// TwinCAT 3 PLC project mini_powermeter_calib
// ProgramVersion: 3.1.4022.7
// libraries:
//   LCLS General, * (SLAC)
//   lcls-twincat-motion, * (SLAC)
//   lcls2-cc-lib, * (SLAC)
//   PMPS, * (SLAC - LCLS)
//   Tc2_Standard, * (Beckhoff Automation GmbH)
//   Tc2_System, * (Beckhoff Automation GmbH)
//   Tc3_Module, * (Beckhoff Automation GmbH)
// project tree:
//   / GlobalTextList.TcGTLO, PlcTask.TcTTO
//   GVLs/ GVL.TcGVL, Main.TcGVL
//   POUs/ FB_AnalogInput_DINT.TcPOU, FB_PPM_PowerMeter_DINT.TcPOU, PRG_MAIN.TcPOU, PRG_IM1_PPM.TcPOU, PRG_IM2_PPM.TcPOU
// real-time tasks:
//   TASK PlcTask: cycle T#10ms, priority 20, ADS port 350
//   TASK VISU_TASK: cycle T#200000us, priority 30, ADS port 351
// motion (NC):
//   TASK NC-Task 1 SAF: cycle T#2ms, priority 4, ADS port 501
//   TASK NC-Task 1 SVB: cycle T#10ms, priority 8, ADS port 511
//   AXIS Axis 1 IM1TST-PPM-MMS (id 1)
//     Dynamic: AccelerationMaximum=200, DecelerationMaximum=200, Acceleration=200, Deceleration=200, Jerk=1000, DelayTime=0.004
//     Velo: Maximum=65
//     MotionControl: Enable=true, Range=0.0005, Time=1
//     TargetPosControl: Range=0.01, Time=1
//     OtherSettings: AllowMotionCmdToSlave=true
//     encoder EncType=29
//       EncPara: ScaleFactorNumerator=5e-05, Offset=-214686.941, MaxCount=#xffffffff, MaxCountHighDWord=#x0000001f
//         SoftEndMinControl: Enable=true, Range=-101.12
//         SoftEndMaxControl: Enable=true, Range=-11
//         Inc: RefSoftSyncMask=#x0000ffff
//     drive DrvType=24
//       Analog: VeloReferenz=100, ScaleFactorActTorque=0.1
//       TimeComp: TaskDelayCycles=1
//     controller CtrType=2
//       CtrPara: PriorControlFactor=1
//         PosDiffControl: Range=10, Time=0.1
//         PID: PosKp=10, PosExtKp=0.01, PosExtVelo=0.0005, DeadBandPosition=0.0001
//         Observer: BandWidth=20
//   AXIS Axis 2 IM2TST-PPM-MMS (id 23)
//     Dynamic: AccelerationMaximum=200, DecelerationMaximum=200, Acceleration=200, Deceleration=200, Jerk=1000, DelayTime=0.004
//     Velo: Maximum=65
//     MotionControl: Enable=true, Range=0.0005, Time=1
//     TargetPosControl: Range=0.01, Time=1
//     OtherSettings: AllowMotionCmdToSlave=true
//     encoder EncType=29
//       EncPara: ScaleFactorNumerator=5e-05, Offset=-214686.941, MaxCount=#xffffffff, MaxCountHighDWord=#x0000001f
//         SoftEndMinControl: Enable=true, Range=-101.12
//         SoftEndMaxControl: Enable=true, Range=-11
//         Inc: RefSoftSyncMask=#x0000ffff
//     drive DrvType=24
//       Analog: VeloReferenz=100, ScaleFactorActTorque=0.1
//       TimeComp: TaskDelayCycles=1
//     controller CtrType=2
//       CtrPara: PriorControlFactor=1
//         PosDiffControl: Range=10, Time=0.1
//         PID: PosKp=10, PosExtKp=0.01, PosExtVelo=0.0005, DeadBandPosition=0.0001
//         Observer: BandWidth=20
// I/O:
//   DEVICE Device 1 (EtherCAT), AmsNetId 172.21.148.90.2.1
//     Term 1 (EK1200) [EK1200-5000 EtherCAT Power supply (2A E-Bus)]
//       Term 2 (EL3602) [EL3602 2Ch. Ana. Input +/-10Volt, Diff. 24bit]
//       Term 3 (EK1122) [EK1122 2 port EtherCAT junction]
//         X1 IM1-PPM (EK1100) [EK1100 EtherCAT Coupler (2A E-Bus)]
//           IM1-EL7041 [EL7041 1Ch. Stepper motor output stage (50V, 5A)]
//           IM1-EL5042 [EL5042 2Ch. BiSS-C Encoder]
//           IM1-EL2004 [EL2004 4Ch. Dig. Output 24V, 0.5A]
//           IM1-EL3314 [EL3314 4Ch. Ana. Input Thermocouple (TC)]
//           IM1-EL3052 [EL3052 2Ch. Ana. Input 4-20mA]
//           IM1-EL3062 [EL3062 2Ch. Ana. Input 0-10V]
//           IM1-EL4004 [EL4004 4Ch. Ana. Output 0-10V, 12bit]
//           IM1-EL9011
//         X2 IM2-PPM (EK1100) [EK1100 EtherCAT Coupler (2A E-Bus)]
//           IM2-EL7041 [EL7041 1Ch. Stepper motor output stage (50V, 5A)]
//           IM2-EL5042 [EL5042 2Ch. BiSS-C Encoder]
//           IM2-EL2004 [EL2004 4Ch. Dig. Output 24V, 0.5A]
//           IM2-EL3314 [EL3314 4Ch. Ana. Input Thermocouple (TC)]
//           IM2-EL3052 [EL3052 2Ch. Ana. Input 4-20mA]
//           IM2-EL3062 [EL3062 2Ch. Ana. Input 0-10V]
//           IM2-EL4004 [EL4004 4Ch. Ana. Output 0-10V, 12bit]
//           IM2-EL9011 [EL9011 End Terminal]
//       Term 4 (EL9011) [EL9011 End Terminal]
// variable links:
//   (this object) <-> Device 1 (EtherCAT)/Term 1 (EK1200)/Term 3 (EK1122)/X1 IM1-PPM (EK1100)/IM1-EL5042
//     Enc/Inputs/In/nComState @bit 1 <-> WcState/InputToggle
//     Enc/Inputs/In/nComState <-> WcState/WcState
//     Enc/Inputs/In/nDataIn1 <-> FB Inputs Channel 1/Position
//     Enc/Inputs/In/nState1 @bit 12 <-> FB Inputs Channel 1/Status/Diag
//     Enc/Inputs/In/nState1 @bit 1 <-> FB Inputs Channel 1/Status/Error
//     Enc/Inputs/In/nState1 @bit 14 <-> FB Inputs Channel 1/Status/Input cycle counter
//     Enc/Inputs/In/nState1 @bit 2 <-> FB Inputs Channel 1/Status/Ready
//     Enc/Inputs/In/nState1 @bit 13 <-> FB Inputs Channel 1/Status/TxPDO State
//     Enc/Inputs/In/nState1 <-> FB Inputs Channel 1/Status/Warning
//   (this object) <-> Device 1 (EtherCAT)/Term 1 (EK1200)/Term 3 (EK1122)/X1 IM1-PPM (EK1100)/IM1-EL7041
//     Drive/Inputs/In/nState1 @bit 3 <-> STM Status/Status/Error
//     Drive/Inputs/In/nState1 @bit 5 <-> STM Status/Status/Moving negative
//     Drive/Inputs/In/nState1 @bit 4 <-> STM Status/Status/Moving positive
//     Drive/Inputs/In/nState1 @bit 1 <-> STM Status/Status/Ready
//     Drive/Inputs/In/nState1 <-> STM Status/Status/Ready to enable
//     Drive/Inputs/In/nState1 @bit 6 <-> STM Status/Status/Torque reduced
//     Drive/Inputs/In/nState1 @bit 2 <-> STM Status/Status/Warning
//     Drive/Inputs/In/nState2 @bit 3 <-> STM Status/Status/Digital input 1
//     Drive/Inputs/In/nState2 @bit 4 <-> STM Status/Status/Digital input 2
//     Drive/Inputs/In/nState2 @bit 5 <-> STM Status/Status/Sync error
//     Drive/Inputs/In/nState2 @bit 7 <-> STM Status/Status/TxPDO Toggle
//     Drive/Inputs/In/nState4 @bit 1 <-> WcState/InputToggle
//     Drive/Inputs/In/nState4 <-> WcState/WcState
//     Drive/Outputs/Out/nCtrl1 <-> STM Control/Control/Enable
//     Drive/Outputs/Out/nCtrl1 @bit 2 <-> STM Control/Control/Reduce torque
//     Drive/Outputs/Out/nCtrl1 @bit 1 <-> STM Control/Control/Reset
//     Drive/Outputs/Out/nDataOut2[0] <-> STM Velocity/Velocity
//   (this object) <-> Device 1 (EtherCAT)/Term 1 (EK1200)/Term 3 (EK1122)/X2 IM2-PPM (EK1100)/IM2-EL5042
//     Enc/Inputs/In/nComState @bit 1 <-> WcState/InputToggle
//     Enc/Inputs/In/nComState <-> WcState/WcState
//     Enc/Inputs/In/nDataIn1 <-> FB Inputs Channel 1/Position
//     Enc/Inputs/In/nState1 @bit 12 <-> FB Inputs Channel 1/Status/Diag
//     Enc/Inputs/In/nState1 @bit 1 <-> FB Inputs Channel 1/Status/Error
//     Enc/Inputs/In/nState1 @bit 14 <-> FB Inputs Channel 1/Status/Input cycle counter
//     Enc/Inputs/In/nState1 @bit 2 <-> FB Inputs Channel 1/Status/Ready
//     Enc/Inputs/In/nState1 @bit 13 <-> FB Inputs Channel 1/Status/TxPDO State
//     Enc/Inputs/In/nState1 <-> FB Inputs Channel 1/Status/Warning
//   (this object) <-> Device 1 (EtherCAT)/Term 1 (EK1200)/Term 3 (EK1122)/X2 IM2-PPM (EK1100)/IM2-EL7041
//     Drive/Inputs/In/nState1 @bit 3 <-> STM Status/Status/Error
//     Drive/Inputs/In/nState1 @bit 5 <-> STM Status/Status/Moving negative
//     Drive/Inputs/In/nState1 @bit 4 <-> STM Status/Status/Moving positive
//     Drive/Inputs/In/nState1 @bit 1 <-> STM Status/Status/Ready
//     Drive/Inputs/In/nState1 <-> STM Status/Status/Ready to enable
//     Drive/Inputs/In/nState1 @bit 6 <-> STM Status/Status/Torque reduced
//     Drive/Inputs/In/nState1 @bit 2 <-> STM Status/Status/Warning
//     Drive/Inputs/In/nState2 @bit 3 <-> STM Status/Status/Digital input 1
//     Drive/Inputs/In/nState2 @bit 4 <-> STM Status/Status/Digital input 2
//     Drive/Inputs/In/nState2 @bit 5 <-> STM Status/Status/Sync error
//     Drive/Inputs/In/nState2 @bit 7 <-> STM Status/Status/TxPDO Toggle
//     Drive/Inputs/In/nState4 @bit 1 <-> WcState/InputToggle
//     Drive/Inputs/In/nState4 <-> WcState/WcState
//     Drive/Outputs/Out/nCtrl1 <-> STM Control/Control/Enable
//     Drive/Outputs/Out/nCtrl1 @bit 2 <-> STM Control/Control/Reduce torque
//     Drive/Outputs/Out/nCtrl1 @bit 1 <-> STM Control/Control/Reset
//     Drive/Outputs/Out/nDataOut2[0] <-> STM Velocity/Velocity
//   mini_powermeter_calib Instance <-> Device 1 (EtherCAT)/Term 1 (EK1200)/Term 2 (EL3602)
//     PlcTask Inputs/PRG_MAIN.fb_pm.iVoltageINT <-> AI Inputs Channel 1/Value
//   mini_powermeter_calib Instance <-> Device 1 (EtherCAT)/Term 1 (EK1200)/Term 3 (EK1122)/X1 IM1-PPM (EK1100)/IM1-EL2004
//     PlcTask Outputs/Main.M1.bBrakeRelease <-> Channel 1/Output
//     PlcTask Outputs/PRG_IM1_PPM.fbIM1.fbGige.bGigePower <-> Channel 2/Output
//   mini_powermeter_calib Instance <-> Device 1 (EtherCAT)/Term 1 (EK1200)/Term 3 (EK1122)/X1 IM1-PPM (EK1100)/IM1-EL3062
//     PlcTask Inputs/PRG_IM1_PPM.fbIM1.fbPowerMeter.iVoltageINT <-> AI Standard Channel 1/Value
//   mini_powermeter_calib Instance <-> Device 1 (EtherCAT)/Term 1 (EK1200)/Term 3 (EK1122)/X1 IM1-PPM (EK1100)/IM1-EL3314
//     PlcTask Inputs/PRG_IM1_PPM.fbIM1.fbPowerMeter.fbThermoCouple.bError <-> TC Inputs Channel 1/Status/Error
//     PlcTask Inputs/PRG_IM1_PPM.fbIM1.fbPowerMeter.fbThermoCouple.bOverrange <-> TC Inputs Channel 1/Status/Overrange
//     PlcTask Inputs/PRG_IM1_PPM.fbIM1.fbPowerMeter.fbThermoCouple.bUnderrange <-> TC Inputs Channel 1/Status/Underrange
//     PlcTask Inputs/PRG_IM1_PPM.fbIM1.fbPowerMeter.fbThermoCouple.iRaw <-> TC Inputs Channel 1/Value
//     PlcTask Inputs/PRG_IM1_PPM.fbIM1.fbYagThermoCouple.bError <-> TC Inputs Channel 2/Status/Error
//     PlcTask Inputs/PRG_IM1_PPM.fbIM1.fbYagThermoCouple.bOverrange <-> TC Inputs Channel 2/Status/Overrange
//     PlcTask Inputs/PRG_IM1_PPM.fbIM1.fbYagThermoCouple.bUnderrange <-> TC Inputs Channel 2/Status/Underrange
//     PlcTask Inputs/PRG_IM1_PPM.fbIM1.fbYagThermoCouple.iRaw <-> TC Inputs Channel 2/Value
//   mini_powermeter_calib Instance <-> Device 1 (EtherCAT)/Term 1 (EK1200)/Term 3 (EK1122)/X1 IM1-PPM (EK1100)/IM1-EL4004
//     PlcTask Outputs/PRG_IM1_PPM.fbIM1.fbGige.iIlluminatorINT <-> AO Outputs Channel 1/Analog output
//   mini_powermeter_calib Instance <-> Device 1 (EtherCAT)/Term 1 (EK1200)/Term 3 (EK1122)/X1 IM1-PPM (EK1100)/IM1-EL7041
//     PlcTask Inputs/Main.M1.bLimitBackwardEnable <-> STM Status/Status/Digital input 2
//     PlcTask Inputs/Main.M1.bLimitForwardEnable <-> STM Status/Status/Digital input 1
//   mini_powermeter_calib Instance <-> Device 1 (EtherCAT)/Term 1 (EK1200)/Term 3 (EK1122)/X2 IM2-PPM (EK1100)/IM2-EL2004
//     PlcTask Outputs/Main.M2.bBrakeRelease <-> Channel 1/Output
//     PlcTask Outputs/PRG_IM2_PPM.fbIM2.fbGige.bGigePower <-> Channel 2/Output
//   mini_powermeter_calib Instance <-> Device 1 (EtherCAT)/Term 1 (EK1200)/Term 3 (EK1122)/X2 IM2-PPM (EK1100)/IM2-EL3062
//     PlcTask Inputs/PRG_IM2_PPM.fbIM2.fbPowerMeter.iVoltageINT <-> AI Standard Channel 1/Value
//   mini_powermeter_calib Instance <-> Device 1 (EtherCAT)/Term 1 (EK1200)/Term 3 (EK1122)/X2 IM2-PPM (EK1100)/IM2-EL3314
//     PlcTask Inputs/PRG_IM2_PPM.fbIM2.fbPowerMeter.fbThermoCouple.bError <-> TC Inputs Channel 1/Status/Error
//     PlcTask Inputs/PRG_IM2_PPM.fbIM2.fbPowerMeter.fbThermoCouple.bOverrange <-> TC Inputs Channel 1/Status/Overrange
//     PlcTask Inputs/PRG_IM2_PPM.fbIM2.fbPowerMeter.fbThermoCouple.bUnderrange <-> TC Inputs Channel 1/Status/Underrange
//     PlcTask Inputs/PRG_IM2_PPM.fbIM2.fbPowerMeter.fbThermoCouple.iRaw <-> TC Inputs Channel 1/Value
//     PlcTask Inputs/PRG_IM2_PPM.fbIM2.fbYagThermoCouple.bError <-> TC Inputs Channel 2/Status/Error
//     PlcTask Inputs/PRG_IM2_PPM.fbIM2.fbYagThermoCouple.bOverrange <-> TC Inputs Channel 2/Status/Overrange
//     PlcTask Inputs/PRG_IM2_PPM.fbIM2.fbYagThermoCouple.bUnderrange <-> TC Inputs Channel 2/Status/Underrange
//     PlcTask Inputs/PRG_IM2_PPM.fbIM2.fbYagThermoCouple.iRaw <-> TC Inputs Channel 2/Value
//   mini_powermeter_calib Instance <-> Device 1 (EtherCAT)/Term 1 (EK1200)/Term 3 (EK1122)/X2 IM2-PPM (EK1100)/IM2-EL4004
//     PlcTask Outputs/PRG_IM2_PPM.fbIM2.fbGige.iIlluminatorINT <-> AO Outputs Channel 1/Analog output
//   mini_powermeter_calib Instance <-> Device 1 (EtherCAT)/Term 1 (EK1200)/Term 3 (EK1122)/X2 IM2-PPM (EK1100)/IM2-EL7041
//     PlcTask Inputs/Main.M2.bLimitBackwardEnable <-> STM Status/Status/Digital input 2
//     PlcTask Inputs/Main.M2.bLimitForwardEnable <-> STM Status/Status/Digital input 1
//   mini_powermeter_calib Instance <-> NC-Task 1 SAF/Axes/Axis 1 IM1TST-PPM-MMS
//     PlcTask Inputs/Main.M1.Axis.NcToPlc <-> Outputs/ToPlc
//     PlcTask Outputs/Main.M1.Axis.PlcToNc <-> Inputs/FromPlc
//   mini_powermeter_calib Instance <-> NC-Task 1 SAF/Axes/Axis 2 IM2TST-PPM-MMS
//     PlcTask Inputs/Main.M2.Axis.NcToPlc <-> Outputs/ToPlc
//     PlcTask Outputs/Main.M2.Axis.PlcToNc <-> Inputs/FromPlc

CONFIGURATION mini_powermeter_calib
    RESOURCE PLC ON TwinCAT3
        TASK PlcTask(INTERVAL := T#10ms, PRIORITY := 20);
        PROGRAM PRG_MAIN WITH PlcTask : PRG_MAIN;
    END_RESOURCE
END_CONFIGURATION

// ---- GVLs/GVL.TcGVL
{attribute 'qualified_only'}
VAR_GLOBAL
    fbArbiter: FB_Arbiter(1);
    fbFastFaultOutput1: FB_HardwareFFOutput := (bAutoReset := TRUE);
END_VAR

// ---- GVLs/Main.TcGVL
{attribute 'qualified_only'}
VAR_GLOBAL
    {attribute 'pytmc' := 'pv: IM1TST:PPM:MMS'}
    {attribute 'TcLinkTo' := '.bLimitForwardEnable  := TIIB[IM1-EL7041]^STM Status^Status^Digital input 1;
                              .bLimitBackwardEnable := TIIB[IM1-EL7041]^STM Status^Status^Digital input 2;
                              .bBrakeRelease        := TIIB[IM1-EL2004]^Channel 1^Output'}
    M1: DUT_MotionStage := (sName := 'IM1TST:PPM:MMS');
    {attribute 'pytmc' := 'pv: IM2TST:PPM:MMS'}
    {attribute 'TcLinkTo' := '.bLimitForwardEnable  := TIIB[IM2-EL7041]^STM Status^Status^Digital input 1;
                              .bLimitBackwardEnable := TIIB[IM2-EL7041]^STM Status^Status^Digital input 2;
                              .bBrakeRelease        := TIIB[IM2-EL2004]^Channel 1^Output'}
    M2: DUT_MotionStage := (sName := 'IM2TST:PPM:MMS');
END_VAR

// ---- POUs/PRG_MAIN.TcPOU
PROGRAM PRG_MAIN
VAR
    {attribute 'pytmc' := '
        pv: TST:WFS:SPM
        io: i
    '}
    fb_pm: FB_PPM_PowerMeter_DINT;
END_VAR

fb_pm();
PRG_IM1_PPM();
PRG_IM2_PPM();

END_PROGRAM

// ---- POUs/FB_PPM_PowerMeter_DINT.TcPOU
FUNCTION_BLOCK FB_PPM_PowerMeter_DINT
VAR
    iVoltageINT AT %I*: DINT;

    {attribute 'pytmc' := '
        pv: VOLT
        io: input
        field: EGU mV
    '}
    fVoltage: LREAL;

    {attribute 'pytmc' := '
        pv: VOLT_BUFFER
        io: input
        field: EGU mV
    '}
    fVoltageBuffer: ARRAY[1..1000] OF LREAL;

    {attribute 'pytmc' := '
        pv: CALIB
        io: input
    '}
    fCalibBase: LREAL;

    {attribute 'pytmc' := '
        pv: CALIB_BUFFER
        io: input
    '}
    fCalibBaseBuffer: ARRAY[1..1000] OF LREAL;

    {attribute 'pytmc' := '
        pv: MJ
        io: input
        field: EGU mJ
    '}
    fCalibMJ: LREAL;

    {attribute 'pytmc' := '
        pv: MJ_BUFFER
        io: input
        field: EGU mJ
    '}
    fCalibMJBuffer: ARRAY[1..1000] OF LREAL;

    {attribute 'pytmc' := '
        pv:
        io: input
    '}
    fbThermoCouple: FB_ThermoCouple;

    {attribute 'pytmc' := '
        pv: CALIB:OFFSET
        io: io
    '}
    fCalibRelOffset: LREAL;

    {attribute 'pytmc' := '
        pv: CALIB:RATIO
        io: io
    '}
    fCalibRelRatio: LREAL;

    {attribute 'pytmc' := '
        pv: CALIB:MJ_RATIO
        io: io
    '}
    fCalibMJRatio: LREAL;

    fbGetPMVoltage: FB_AnalogInput_DINT;
    fbVoltageBuffer: FB_LREALBuffer;
    fbCalibBaseBuffer: FB_LREALBuffer;
    fbCalibMJBuffer: FB_LREALBuffer;
END_VAR

fbThermoCouple();

// Convert the terminal's integer into a value in millivolts
fbGetPMVoltage(
    iRaw := iVoltageINT,
    iTermBits := 24,
    fTermMax := 10000,
    fTermMin := 0,
    fReal => fVoltage);

// Power meter calibration
fCalibBase := (fVoltage + fCalibRelOffset) * fCalibRelRatio;
fCalibMJ := fCalibBase * fCalibMJRatio;

// Buffer the full-rate Voltage and calibrated MJ values
fbVoltageBuffer(
    bExecute := TRUE,
    fInput := fVoltage,
    arrOutput => fVoltageBuffer);
fbCalibBaseBuffer(
    bExecute := TRUE,
    fInput := fCalibBase,
    arrOutput => fCalibBaseBuffer);
fbCalibMJBuffer(
    bExecute := TRUE,
    fInput := fCalibMJ,
    arrOutput => fCalibMJBuffer);

END_FUNCTION_BLOCK

// ---- POUs/FB_AnalogInput_DINT.TcPOU
{attribute 'no_check'}
FUNCTION_BLOCK FB_AnalogInput_DINT
(*
    Converts the integer from an analog input terminal to a real unit value (e.g., volts)
    2019-10-09 Zachary Lentz
*)
VAR_INPUT
    // Connect this input to the terminal
    iRaw AT %I*: DINT;
    // The number of bits correlated with the terminal's max value. This is not necessarily the resolution parameter.
    iTermBits: UINT;
    // The fReal value correlated with the terminal's max value
    fTermMax: LREAL;
    // The fReal value correlated with the terminal's min value
    fTermMin: LREAL;
END_VAR
VAR_OUTPUT
    // The real value read from the output
    fReal: LREAL;
END_VAR
VAR
    fScale: LREAL;
END_VAR

IF fScale = 0 AND fTermMax > fTermMin THEN
    fScale := (EXPT(2, iTermBits) - 1) / (fTermMax - fTermMin);
END_IF
IF fScale <> 0 THEN
    fReal := iRaw / fScale + fTermMin;
END_IF

END_FUNCTION_BLOCK

// ---- POUs/PRG_IM1_PPM.TcPOU
PROGRAM PRG_IM1_PPM
VAR
    {attribute 'pytmc' := '
        pv: IM1TST:PPM
        io: io
    '}
    {attribute 'TcLinkTo' := '.fbGige.iIlluminatorINT := TIIB[IM1-EL4004]^AO Outputs Channel 1^Analog output;
                              .fbGige.bGigePower := TIIB[IM1-EL2004]^Channel 2^Output;
                              .fbPowerMeter.iVoltageINT := TIIB[IM1-EL3062]^AI Standard Channel 1^Value;
                              .fbPowerMeter.fbThermoCouple.bError := TIIB[IM1-EL3314]^TC Inputs Channel 1^Status^Error;
                              .fbPowerMeter.fbThermoCouple.bUnderrange := TIIB[IM1-EL3314]^TC Inputs Channel 1^Status^Underrange;
                              .fbPowerMeter.fbThermoCouple.bOverrange := TIIB[IM1-EL3314]^TC Inputs Channel 1^Status^Overrange;
                              .fbPowerMeter.fbThermoCouple.iRaw := TIIB[IM1-EL3314]^TC Inputs Channel 1^Value;
                              .fbYagThermoCouple.bError := TIIB[IM1-EL3314]^TC Inputs Channel 2^Status^Error;
                              .fbYagThermoCouple.bUnderrange := TIIB[IM1-EL3314]^TC Inputs Channel 2^Status^Underrange;
                              .fbYagThermoCouple.bOverrange := TIIB[IM1-EL3314]^TC Inputs Channel 2^Status^Overrange;
                              .fbYagThermoCouple.iRaw := TIIB[IM1-EL3314]^TC Inputs Channel 2^Value'}
    fbIM1: FB_PPM;

    bInit: BOOL := TRUE;
END_VAR


IF bInit THEN
    fbIM1.nTransitionAssertionID := 16#2110;
    fbIM1.nUnknownAssertionID := 16#2119;

    fbIM1.stOut.fPosition := -11;
    fbIM1.stOut.bUseRawCounts := FALSE;
    fbIM1.stOut.nRequestAssertionID := 16#2111;
    fbIM1.stOut.stBeamParams := PMPS_GVL.cstFullBeam;
    fbIM1.stOut.bValid := TRUE;

    fbIM1.stPower.fPosition := -47.59;
    fbIM1.stPower.bUseRawCounts := FALSE;
    fbIM1.stPower.nRequestAssertionID := 16#2112;
    fbIM1.stPower.stBeamParams := PMPS_GVL.cstFullBeam;
    // For now, leave this restriction out (doesn't even take beam yet)
    // fbIM1.stPower.stBeamParams := F_eVExcludeRange(1, 5000);
    fbIM1.stPower.bValid := TRUE;

    fbIM1.stYag1.fPosition := -71.69;
    fbIM1.stYag1.bUseRawCounts := FALSE;
    fbIM1.stYag1.nRequestAssertionID := 16#2113;
    fbIM1.stYag1.stBeamParams := PMPS_GVL.cstFullBeam;
    // For now, do not have restrictions on this YAG. Eventually we want to add exclusion ranges where we need to limit transmission to 0.1 (10%) within those ranges. Currently we do not have transmission control via PMPS on LFE.
    // fbIM1.stYag1.stBeamParams.neVRange := F_eVExcludeRange(2100, 3800) AND F_eVExcludeRange(16900, 24000);
    fbIM1.stYag1.bValid := TRUE;

    fbIM1.stYag2.fPosition := -97.70;
    fbIM1.stYag2.bUseRawCounts := FALSE;
    fbIM1.stYag2.nRequestAssertionID := 16#2114;
    fbIM1.stYag2.stBeamParams := PMPS_GVL.cstFullBeam;
    // For now, do not have restrictions on this YAG. Eventually we want to add exclusion ranges where we need to limit transmission to 0.1 (10%) within those ranges. Currently we do not have transmission control via PMPS on LFE.
    // fbIM1.stYag2.stBeamParams.neVRange := F_eVExcludeRange(2100, 3800) AND F_eVExcludeRange(16900, 24000);
    fbIM1.stYag2.bValid := TRUE;

    bInit := FALSE;
END_IF

fbIM1(
    fbArbiter := GVL.fbArbiter,
    fbFFHWO := GVL.fbFastFaultOutput1,
    stYStage := Main.M1);

END_PROGRAM

// ---- POUs/PRG_IM2_PPM.TcPOU
PROGRAM PRG_IM2_PPM
VAR
    {attribute 'pytmc' := '
        pv: IM2TST:PPM
        io: io
    '}
    {attribute 'TcLinkTo' := '.fbGige.iIlluminatorINT := TIIB[IM2-EL4004]^AO Outputs Channel 1^Analog output;
                              .fbGige.bGigePower := TIIB[IM2-EL2004]^Channel 2^Output;
                              .fbPowerMeter.iVoltageINT := TIIB[IM2-EL3062]^AI Standard Channel 1^Value;
                              .fbPowerMeter.fbThermoCouple.bError := TIIB[IM2-EL3314]^TC Inputs Channel 1^Status^Error;
                              .fbPowerMeter.fbThermoCouple.bUnderrange := TIIB[IM2-EL3314]^TC Inputs Channel 1^Status^Underrange;
                              .fbPowerMeter.fbThermoCouple.bOverrange := TIIB[IM2-EL3314]^TC Inputs Channel 1^Status^Overrange;
                              .fbPowerMeter.fbThermoCouple.iRaw := TIIB[IM2-EL3314]^TC Inputs Channel 1^Value;
                              .fbYagThermoCouple.bError := TIIB[IM2-EL3314]^TC Inputs Channel 2^Status^Error;
                              .fbYagThermoCouple.bUnderrange := TIIB[IM2-EL3314]^TC Inputs Channel 2^Status^Underrange;
                              .fbYagThermoCouple.bOverrange := TIIB[IM2-EL3314]^TC Inputs Channel 2^Status^Overrange;
                              .fbYagThermoCouple.iRaw := TIIB[IM2-EL3314]^TC Inputs Channel 2^Value'}
    fbIM2: FB_PPM;

    bInit: BOOL := TRUE;
END_VAR


IF bInit THEN
    fbIM2.nTransitionAssertionID := 16#2110;
    fbIM2.nUnknownAssertionID := 16#2119;

    fbIM2.stOut.fPosition := -11;
    fbIM2.stOut.bUseRawCounts := FALSE;
    fbIM2.stOut.nRequestAssertionID := 16#2111;
    fbIM2.stOut.stBeamParams := PMPS_GVL.cstFullBeam;
    fbIM2.stOut.bValid := TRUE;

    fbIM2.stPower.fPosition := -47.59;
    fbIM2.stPower.bUseRawCounts := FALSE;
    fbIM2.stPower.nRequestAssertionID := 16#2112;
    fbIM2.stPower.stBeamParams := PMPS_GVL.cstFullBeam;
    // For now, leave this restriction out (doesn't even take beam yet)
    // fbIM2.stPower.stBeamParams := F_eVExcludeRange(1, 5000);
    fbIM2.stPower.bValid := TRUE;

    fbIM2.stYag1.fPosition := -71.69;
    fbIM2.stYag1.bUseRawCounts := FALSE;
    fbIM2.stYag1.nRequestAssertionID := 16#2113;
    fbIM2.stYag1.stBeamParams := PMPS_GVL.cstFullBeam;
    // For now, do not have restrictions on this YAG. Eventually we want to add exclusion ranges where we need to limit transmission to 0.1 (10%) within those ranges. Currently we do not have transmission control via PMPS on LFE.
    // fbIM2.stYag1.stBeamParams.neVRange := F_eVExcludeRange(2100, 3800) AND F_eVExcludeRange(16900, 24000);
    fbIM2.stYag1.bValid := TRUE;

    fbIM2.stYag2.fPosition := -97.70;
    fbIM2.stYag2.bUseRawCounts := FALSE;
    fbIM2.stYag2.nRequestAssertionID := 16#2114;
    fbIM2.stYag2.stBeamParams := PMPS_GVL.cstFullBeam;
    // For now, do not have restrictions on this YAG. Eventually we want to add exclusion ranges where we need to limit transmission to 0.1 (10%) within those ranges. Currently we do not have transmission control via PMPS on LFE.
    // fbIM2.stYag2.stBeamParams.neVRange := F_eVExcludeRange(2100, 3800) AND F_eVExcludeRange(16900, 24000);
    fbIM2.stYag2.bValid := TRUE;

    bInit := FALSE;
END_IF

fbIM2(
    fbArbiter := GVL.fbArbiter,
    fbFFHWO := GVL.fbFastFaultOutput1,
    stYStage := Main.M2);

END_PROGRAM

// ---- GlobalTextList.TcGTLO
TEXTLIST GlobalTextList
  670 = 'Measuring %f mV'
  168 = 'Voltage is %f mV'
END_TEXTLIST
